TYPE INTERNAL ST_Entry :
STRUCT
	iSignal		: I_SignalNode;
	iReceiver	: I_ReceiverNode;
END_STRUCT
END_TYPE

(* stored: Version 1.1.0.1
   DUT ST_Entry: Id {c7a7d29f-efe7-4297-b94b-aa4eb559cb25} *)
